PROGRAM main
  VAR
    MOTOR_ON_PB AT %IX0.0 : BOOL;
    EMERGENCY_PB AT %IX0.1 : BOOL;
    MOTOR_STOP_PB AT %IX0.2 : BOOL;
    TEST_IN_01 AT %IX0.3 : BOOL;
    TEST_IN_02 AT %IX0.4 : BOOL;
    MOTOR_ON AT %QX0.0 : BOOL;
    GREEN_LAMP AT %QX0.1 : BOOL;
    RED_LAMP AT %QX0.2 : BOOL;
    ORANGE_LAMP AT %QX0.3 : BOOL;
    TEST_OUT_1 AT %QX0.4 : BOOL;
    TEST_OUT_2 AT %QX0.5 : BOOL;
  END_VAR

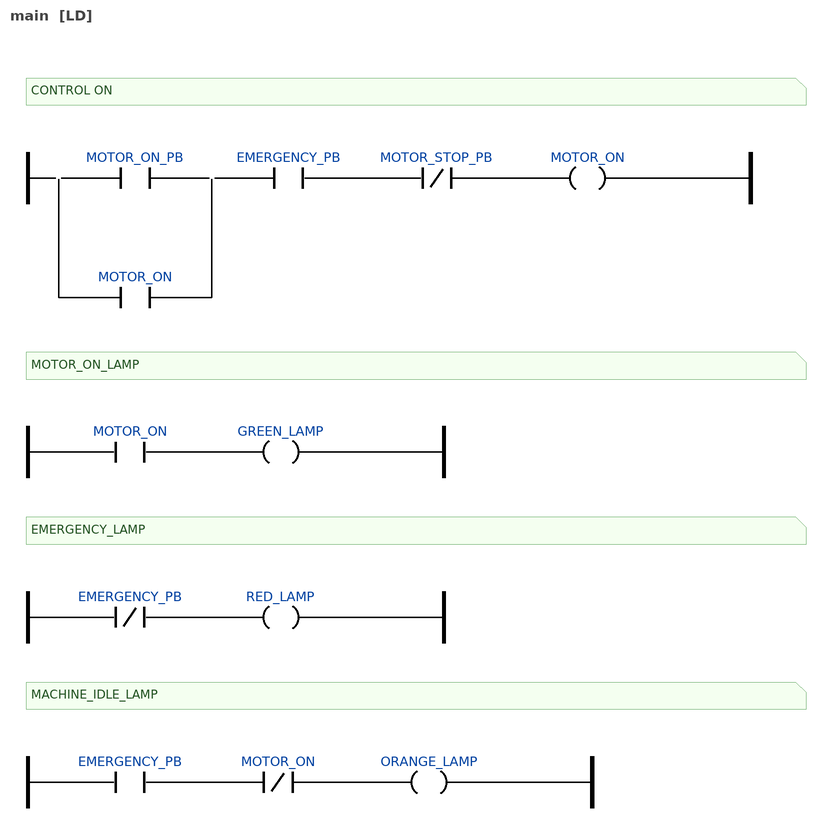
(* LD diagram, written out as Structured Text *)
(* CONTROL ON *)
MOTOR_ON := (MOTOR_ON_PB OR MOTOR_ON) AND EMERGENCY_PB AND NOT MOTOR_STOP_PB;
(* MOTOR_ON_LAMP *)
GREEN_LAMP := MOTOR_ON;
(* EMERGENCY_LAMP *)
RED_LAMP := NOT EMERGENCY_PB;
(* MACHINE_IDLE_LAMP *)
ORANGE_LAMP := EMERGENCY_PB AND NOT MOTOR_ON;
END_PROGRAM
